// Represents the months of the year.
{attribute 'qualified_only'}
{attribute 'to_string'}
TYPE E_Month :
(
	_ := 0, // Uninitialised or default value, representing an undefined month.
	January,
	February,
	March,
	April,
	May, 
	June, 
	July,
	August,
	September,
	October,
	November,
	December
)UINT;
END_TYPE

(* stored: Version 1.1.0.1
   EnumerationTextList E_Month: Id {dc82db6b-894d-02eb-2473-80081c97c815} *)
